// TIA Portal V17 export
// export: Created 2025-06-26T06:49:21.2301875Z, ExportSetting WithDefaults, DisplayName Totally Integrated Automation Portal, DisplayVersion V17 Update 8, DisplayName TIA Portal Openness, DisplayVersion V17 Update 8, DisplayName TIA Portal Version Control Interface, DisplayVersion V17, DisplayName STEP 7 Professional, DisplayVersion V17 Update 8, DisplayName STEP 7 Safety, DisplayVersion V17 Update 6, DisplayName WinCC Advanced, DisplayVersion V17 Update 8
DATA_BLOCK "DB_Cloud"   // DB200
{ S7_Optimized_Access := 'TRUE' }
VERSION : 0.1
// stored: AutoNumber false, DBAccessibleFromOPCUA true, IsOnlyStoredInLoadMemory false, IsRetainMemResEnabled false, IsWriteProtectedInAS false, MemoryReserve 0
   VAR
      HBL_TT_502 : Real;
      HBL_PT_503 : Real;
      HBL_TT_504 : Real;
      HBL_LT_510 : Real;
      HBL_PT_511 : Real;
      HBL_TT_512 : Real;
      HBL_TT_516 : Real;
      HBL_PT_517 : Real;
      HBL_TT_518 : Real;
      HBL_PT_519 : Real;
      HBL_FT_520 : Real;
      HBL_TT_530 : Real;
      HBL_PT_531 : Real;
      HBL_TT_532 : Real;
      HBL_TT_533 : Real;
      HBL_PT_534 : Real;
      HBL_AT_535 : Real;
      HBL_TT_540 : Real;
      HBL_PT_541 : Real;
      HBL_TT_542 : Real;
      HBL_TT_543 : Real;
      HBL_PT_544 : Real;
      HBL_AT_545 : Real;
      HBL_TT_546 : Real;
      HBL_PT_547 : Real;
      HBL_TT_571 : Real;
      HBL_PT_572 : Real;
      HBL_TT_573 : Real;
      HBL_LT_610 : Real;
      HBL_TT_611 : Real;
      HBL_PT_612 : Real;
      HBL_CT_615 : Real;
      HBL_PT_618 : Real;
      HBL_PT_635 : Real;
      HBL_PT_636 : Real;
      HBL_LT_650 : Real;
      HBL_PT_651 : Real;
      HBL_PT_701 : Real;
      HBL_PT_702 : Real;
      HBL_PT_703 : Real;
      CPC_LT_870 : Real;
      CPC_TT_871 : Real;
      CPC_PT_872 : Real;
      CPC_PT_862 : Real;
      HBL_TT_901 : Real;
      HBL_PT_902 : Real;
      HBL_TT_03 : Real;
      HBL_TT_16 : Real;
      HBL_TT_17 : Real;
      HBL_TT_18 : Real;
      HBL_TT_20 : Real;
      HBL_TT_21 : Real;
      HBL_TT_22 : Real;
      HBL_TT_23 : Real;
      HBL_TT_24 : Real;
      HBL_TT_25 : Real;
      HBL_TT_26 : Real;
      HBL_TT_27 : Real;
      HBL_PT_05 : Real;
      HBL_PT_06 : Real;
      HBL_PT_17 : Real;
      HBL_CT_01 : Real;
      HBL_CT_03 : Real;
      SSC_TT_01 : Real;
      SSC_TT_02 : Real;
      SSC_TT_03 : Real;
      SSC_TT_04 : Real;
      SSC_PIT_01 : Real;
      SSC_PDT_01 : Real;
      SSC_LT_01 : Real;
      HBL_VT_01 : Real;
      HBL_TT_36 : Real;
      Compressor_CrankcaseSaturationTemperature : Real;
      Compressor_CrankcaseSuperheat : Real;
      Compressor_VolumetricEfficiency : Real;
      Compressor_IsentropicEfficiency : Real;
      Compressor_Massflow : Real;
      HeatSink_DeltaT : Real;
      HeatSink_Pinch : Real;
      HeatSink_HeatRate : Real;
      HeatSink_DeltaP : Real;
      HeatSink_Massflow : Real;
      HeatSource_DeltaT : Real;
      HeatSource_Pinch : Real;
      HeatSource_HeatRate : Real;
      HeatSource_DeltaP : Real;
      HeatSource_TemperatureRateOfChange : Real;
      HeatSource_Massflow : Real;
      HighPressPart_CompressorSaturationTemperature : Real;
      HighPressPart_CompressorSuperheat : Real;
      HighPressPart_CondenserSaturationTemperature : Real;
      HighPressPart_CondenserSubcooling : Real;
      HighPressPart_ExpansionValveSubcooling : Real;
      HighPressPart_CondenserDeltaP : Real;
      LowPressPart_EvaporatorSuperheat : Real;
      LowPressPart_CompressorSuperheat : Real;
      LowPressPart_EvaporatorSaturationTemperature : Real;
      LowPressPart_CompressorSaturationTemperature : Real;
      System_Quality : Real;
      System_COP : Real;
      System_ElectricalPower : Real;
      System_TemperatureLift : Real;
      System_MotorEfficiency : Real;
      System_FMEP : Real;
      Auxiliary_ShaftSealDeltaT : Real;
      Auxiliary_CPCPumpDeltaP : Real;
      Misc_OilFilterDeltaP : Real;
      HBL_FS_01 : Bool;
      HBL_FS_02 : Bool;
      HBL_LS_632 : Bool;
      HBL_LS_633 : Bool;
      CPC_LS_864 : Bool;
      VPNUserConnected : Bool;
      HBL_EC_01 : Bool;
      HBL_EC_02 : Bool;
      HBL_HV_630 : Bool;
      HBL_HV_860 : Bool;
      HBL_HV_861 : Bool;
      SSC_P_01 : Bool;
      SSC_F_01 : Bool;
      SSC_P_02 : Bool;
      CPC_P_01 : Bool;
      HBL_HV_631 : Bool;
      HBL_SC_01_A1 : Real;
      HBL_SC_01_A2 : Real;
      HBL_SC_01_A3 : Real;
      HBL_SC_02_A1 : Real;
      HBL_SC_02_A2 : Real;
      HBL_SC_02_A3 : Real;
      HBL_SC_03_A1 : Real;
      HBL_SC_03_A2 : Real;
      HBL_SC_03_A3 : Real;
      HBL_SC_10_A1 : Real;
      HBL_SC_10_A2 : Real;
      HBL_SC_10_A3 : Real;
      HBL_HCV_576_A1 : Real;
      HBL_HCV_578_A1 : Real;
      HBL_HCV_577_A1 : Real;
      HBL_HCV_579_A1 : Real;
      HBL_HCV_515_A1 : Real;
      HBL_HCV_575_A1 : Real;
      HBL_HCV_616_A1 : Real;
      HBL_HCV_700_A1 : Real;
      HBL_HCV_514_A1 : Real;
      HBL_HCV_548_A1 : Real;
      ClientID : String;
      RunningTimeHours : Int;
      RunningTimeMinutes : Int;
      RunningTimeSeconds : Int;
      MachineState : Int;
   END_VAR
BEGIN
END_DATA_BLOCK
